// TIA Portal V19 export
TYPE "LEXCHANGETRAY_typeConstraintRollerIoSignalInterface"
// configuration: LEXCHANGETRAY_typeConstraintRollerIoSignalConfigeration
// commands: LEXCHANGETRAY_typeConstraintRollerIoSignalManualCommands
// monitoring: LEXCHANGETRAY_typeConstraintRollerIoSignalProcessValues
// stored: Access Published
   STRUCT
      configuration : "LEXCHANGETRAY_typeConstraintRollerIoSignalConfigeration";
      commands { S7_SetPoint := 'True'} : "LEXCHANGETRAY_typeConstraintRollerIoSignalManualCommands";
      monitoring { S7_SetPoint := 'True'} : "LEXCHANGETRAY_typeConstraintRollerIoSignalProcessValues";
   END_STRUCT;
END_TYPE
